FUNCTION_BLOCK FB_Chamber1Ep1PrepareWaferTransfer EXTENDS FB_CompositeServiceBase
VAR
	_Step : E_Chamber1Ep1PrepareWaferTransferStep;
	_CommandSubmitted : BOOL;
	_LiftPinMoveParam : ST_Chamber1LiftPinAxisMoveAbsParam;
	_VacuumOffParam : ST_EmptyServiceParam;
END_VAR

M_UpdateCompositeService();

METHOD PROTECTED H_DeclareServices
M_AddDependency(ServiceId := E_Chamber1ServiceId.LiftPinAxisMoveAbs);
M_AddDependency(ServiceId := E_Chamber1ServiceId.VacuumOff);
END_METHOD

METHOD PROTECTED H_GetExecuteSubState : UDINT
H_GetExecuteSubState := TO_UDINT(_Step);
END_METHOD

METHOD PROTECTED H_GetExecuteSubStateName : STRING(80)
H_GetExecuteSubStateName := TO_STRING(_Step);
END_METHOD

METHOD PROTECTED H_OnCompositeExecute : RobustSolution_BATW.E_PackMLHookResult
VAR_INPUT
	bFirstScan	: BOOL;
END_VAR
VAR
	SubmitResult : E_ServiceCallSubmitResult;
	CommandState : E_ServiceInternalCommandState;
	Snapshot : ST_ServiceExecutionSnapshot;
END_VAR
H_OnCompositeExecute := E_PackMLHookResult.Busy;

IF bFirstScan THEN
	_Step := E_Chamber1Ep1PrepareWaferTransferStep.MoveLiftPinAxis;
	_CommandSubmitted := FALSE;

	_LiftPinMoveParam.Position := 70.0;
	_LiftPinMoveParam.Velocity := 20.0;
	_LiftPinMoveParam.Acceleration := 0.0;
	_LiftPinMoveParam.Deceleration := 0.0;
END_IF

CASE _Step OF
	E_Chamber1Ep1PrepareWaferTransferStep.MoveLiftPinAxis:
		IF NOT _CommandSubmitted THEN
			SubmitResult := M_StartDependency(
				ServiceId := E_Chamber1ServiceId.LiftPinAxisMoveAbs,
				Parameters := _LiftPinMoveParam);

			IF SubmitResult = E_ServiceCallSubmitResult.Queued THEN
				_CommandSubmitted := TRUE;
			ELSIF SubmitResult <> E_ServiceCallSubmitResult.Busy THEN
				M_FailSequence(
					ErrorCode := E_CompositeServiceErrorCode.InternalCallSubmitFailed,
					FailedServiceId := E_Chamber1ServiceId.LiftPinAxisMoveAbs,
					SourceErrorId := TO_UDINT(SubmitResult),
					Message := 'LiftPinAxis MoveAbs Start could not be queued.');
			END_IF
			RETURN;
		END_IF

		CommandState := M_GetDependencyCommandState(
			ServiceId := E_Chamber1ServiceId.LiftPinAxisMoveAbs);
		IF CommandState = E_ServiceInternalCommandState.Rejected THEN
			M_FailSequence(
				ErrorCode := E_CompositeServiceErrorCode.InternalCommandRejected,
				FailedServiceId := E_Chamber1ServiceId.LiftPinAxisMoveAbs,
				SourceErrorId := TO_UDINT(E_PackMLCommand.Start),
				Message := 'LiftPinAxis MoveAbs Start was rejected.');
		ELSIF (CommandState = E_ServiceInternalCommandState.Cancelled)
			OR (CommandState = E_ServiceInternalCommandState.None) THEN
			M_FailSequence(
				ErrorCode := E_CompositeServiceErrorCode.InvalidSequenceState,
				FailedServiceId := E_Chamber1ServiceId.LiftPinAxisMoveAbs,
				SourceErrorId := TO_UDINT(CommandState),
				Message := 'LiftPinAxis MoveAbs command state was lost.');
		ELSIF (CommandState = E_ServiceInternalCommandState.Accepted)
			AND M_GetDependencyServiceSnapshot(
				ServiceId := E_Chamber1ServiceId.LiftPinAxisMoveAbs,
				Snapshot => Snapshot)
			AND (Snapshot.PackMLOut.eStateCurrent = E_PackMLState.Complete) THEN
			_Step := E_Chamber1Ep1PrepareWaferTransferStep.VacuumOff;
			_CommandSubmitted := FALSE;
		END_IF

	E_Chamber1Ep1PrepareWaferTransferStep.VacuumOff:
		IF NOT _CommandSubmitted THEN
			SubmitResult := M_StartDependency(
				ServiceId := E_Chamber1ServiceId.VacuumOff,
				Parameters := _VacuumOffParam);

			IF SubmitResult = E_ServiceCallSubmitResult.Queued THEN
				_CommandSubmitted := TRUE;
			ELSIF SubmitResult <> E_ServiceCallSubmitResult.Busy THEN
				M_FailSequence(
					ErrorCode := E_CompositeServiceErrorCode.InternalCallSubmitFailed,
					FailedServiceId := E_Chamber1ServiceId.VacuumOff,
					SourceErrorId := TO_UDINT(SubmitResult),
					Message := 'VacuumOff Start could not be queued.');
			END_IF
			RETURN;
		END_IF

		CommandState := M_GetDependencyCommandState(
			ServiceId := E_Chamber1ServiceId.VacuumOff);
		IF CommandState = E_ServiceInternalCommandState.Rejected THEN
			M_FailSequence(
				ErrorCode := E_CompositeServiceErrorCode.InternalCommandRejected,
				FailedServiceId := E_Chamber1ServiceId.VacuumOff,
				SourceErrorId := TO_UDINT(E_PackMLCommand.Start),
				Message := 'VacuumOff Start was rejected.');
		ELSIF (CommandState = E_ServiceInternalCommandState.Cancelled)
			OR (CommandState = E_ServiceInternalCommandState.None) THEN
			M_FailSequence(
				ErrorCode := E_CompositeServiceErrorCode.InvalidSequenceState,
				FailedServiceId := E_Chamber1ServiceId.VacuumOff,
				SourceErrorId := TO_UDINT(CommandState),
				Message := 'VacuumOff command state was lost.');
		ELSIF (CommandState = E_ServiceInternalCommandState.Accepted)
			AND M_GetDependencyServiceSnapshot(
				ServiceId := E_Chamber1ServiceId.VacuumOff,
				Snapshot => Snapshot)
			AND (Snapshot.PackMLOut.eStateCurrent = E_PackMLState.Complete) THEN
			_Step := E_Chamber1Ep1PrepareWaferTransferStep.Finish;
			_CommandSubmitted := FALSE;
		END_IF

	E_Chamber1Ep1PrepareWaferTransferStep.Finish:
		H_OnCompositeExecute := E_PackMLHookResult.Done;

	ELSE
		M_FailSequence(
			ErrorCode := E_CompositeServiceErrorCode.InvalidSequenceState,
			FailedServiceId := ServiceId,
			SourceErrorId := TO_UDINT(_Step),
			Message := 'Endpoint1PrepareSendWafer entered an invalid sequence step.');
END_CASE
END_METHOD

END_FUNCTION_BLOCK

(* stored: Version 1.1.0.1, ProductVersion 3.1.4026.18
   POU FB_Chamber1Ep1PrepareWaferTransfer: Id {31c0f8a3-2bb7-4853-987f-7b1795d30426}, SpecialFunc None
   Folder HookMethod: Id {858d5fe9-2c92-497c-8c1b-6833d260548b}
   Method H_DeclareServices: Id {1979dc54-f44c-43aa-9c15-89ebd2fc31b9}
   Method H_GetExecuteSubState: Id {12ac4626-2cd6-4b4d-bd14-30262f3181af}
   Method H_GetExecuteSubStateName: Id {35243858-965b-4837-a7ce-4e8151da400b}
   Method H_OnCompositeExecute: Id {6e0866a2-2b89-4e5d-a7f0-96d53557ce83} *)
